Staubli VAL3: getWordAt.pgx

public program getWordAt(num x_nByteIndex, num& x_nBuffer[], num& x_nRes)
begin

  x_nRes=x_nBuffer[x_nByteIndex]*power(2,8)+x_nBuffer[x_nByteIndex+1]

end
